// TIA Portal V20 export
FUNCTION "FC_ChillerMain" : Void   // FC540, SCL
{ S7_Optimized_Access := 'TRUE' }
// stored: AutoNumber false, SetENOAutomatically false
BEGIN
   REGION Description header 
       //==================================================================================
       // POSALUX Swiss SA / (C) Copyright 2025
       //----------------------------------------------------------------------------------
       // Title: FC_Chiller_Main
       // Comment/Function:
       // Author: Fabien Waldt
       // Engineering: TIA Portal v19
       //----------------------------------------------------------------------------------
       // Change log table:
       // Version  | Date     | Expert in charge | Changes applied
       // ---------|----------|------------------|------------------------------------
       // 00.00.01 | 20250904 | FWA              | First released version
       // ==================================================================================
   END_REGION

   REGION Option Chiller : TERMOTEK
       IF "DB_MachineOptions".Chiller.Termotek THEN
           "DB_ChillerTermotek"();
       END_IF;
   END_REGION

   REGION Option Chiller : SMC
       IF "DB_MachineOptions".Chiller.SMC THEN
           "DB_ChillerSMC"();
       END_IF;
   END_REGION
END_FUNCTION
